{attribute 'qualified_only'}
{attribute 'strict'}
{attribute 'to_string'}
TYPE ParserMethod :
(
    ReadFile,
    WriteFile
);
END_TYPE

(* stored: Version 1.1.0.1, ProductVersion 3.1.4024.4
   DUT ParserMethod: Id {d0c0a20a-2911-4eb0-bc46-c097d88e62c9} *)
